{attribute 'linkalways'} 
{attribute 'no_explicit_call' := 'This FB is a CLASS and must be accessed using methods or properties'}
{attribute 'enable_dynamic_creation'}
FUNCTION_BLOCK Node_F_VN_AppendToContainer_TcVnVector4_INT EXTENDS VisionNode
VAR
    aElement : _TcVnVector4_INT;
    ipContainer : _ITcVnContainer;
    hrPrev : _HRESULT(S_OK);
	hresult : _HRESULT(S_OK);
END_VAR

METHOD PUBLIC  Clone : I_Node
VAR
	pNode : POINTER TO Node_F_VN_AppendToContainer_TcVnVector4_INT;
END_VAR
pNode := __NEW(Node_F_VN_AppendToContainer_TcVnVector4_INT);
Clone := pNode^;
END_METHOD

METHOD FB_init : BOOL
VAR_INPUT
	bInitRetains : BOOL; // if TRUE, the retain variables are initialized (warm start / cold start)
	bInCopyCode : BOOL;  // if TRUE, the instance afterwards gets moved into the copy code (online change)
END_VAR
AddInput('aElement', aElement);
AddInput('ipContainer', ipContainer);
AddInput('hrPrev', hrPrev);
AddOutput('ipContainer', ipContainer);
AddOutput('hresult',hresult);
END_METHOD

METHOD PROTECTED OnExecute : HRESULT
hresult.Value := F_VN_AppendToContainer_TcVnVector4_INT(
    aElement := aElement.Value,
	ipContainer := ipContainer.Value,
	hrPrev:= hrPrev.Value);
END_METHOD

METHOD PUBLIC PreExecutionCheck
VAR_INPUT
	Check : I_PreExecutionChecks;
END_VAR
Check.IsTrue(ipContainer.IsValid, 'ipContainer must be a valid container');
END_METHOD

END_FUNCTION_BLOCK

(* stored: Version 1.1.0.1, ProductVersion 3.1.4024.13
   POU Node_F_VN_AppendToContainer_TcVnVector4_INT: Id {8015d29a-0a57-4c58-a2d8-3cbc2976c391}, SpecialFunc None
   Folder Constructor: Id {81985fb8-35ce-4f88-af53-8b8a01503c25}
   Method Clone: Id {305b2aa6-d289-4b57-a6b0-804028364727}
   Method FB_init: Id {56e0be4c-4401-4ab8-9e96-bf88c94b4299}
   Method OnExecute: Id {4dc6c32b-c293-40cb-8837-6e861ab42de3}
   Method PreExecutionCheck: Id {6bc64c07-2c46-4d17-95e4-f80f40d42f1e} *)
